(* IEC 61131-3 sources: repolevel_ST_code_completion/real_groud_truth最新/repoeval_four-level_elevator_control/full_result, 3 files *)

(* ---- F_CheckJobInDirection.st ---- *)
FUNCTION F_CheckJobInDirection : BOOL
VAR_INPUT
	nStartFloor		:	USINT;		//起始楼层
	nEndFloor		:	USINT;		//结束楼层
	bIncreasing		:	BOOL;		//TRUE=向上检查（递增），FALSE=向下检查（递减）
END_VAR

VAR
	i				:	USINT;		//循环变量
	bJobExists		:	BOOL;		//是否存在任务
END_VAR

// 初始化任务存在标志
bJobExists := FALSE;

// 根据检查方向进行任务检查
IF bIncreasing THEN
	// 向上检查任务
	FOR i := nStartFloor TO nEndFloor DO
		IF IGoFloor[i] OR IFloorUp[i] THEN
			bJobExists := TRUE;
			EXIT; // 找到任务后退出循环
		END_IF
	END_FOR;
ELSE
	// 向下检查任务
	FOR i := nStartFloor TO nEndFloor BY -1 DO
		IF IGoFloor[i] OR IFloorDown[i] THEN
			bJobExists := TRUE;
			EXIT; // 找到任务后退出循环
		END_IF
	END_FOR;
END_IF;

// 返回任务存在标志
RETURN bJobExists;
END_FUNCTION

(* ---- F_ClearFloorStop.st ---- *)
FUNCTION F_ClearFloorStop
VAR_INPUT
	nFloor			:	USINT;		//楼层号
	bClearUpStop	:	BOOL;		//是否清除上升停靠标志
	bClearDownStop	:	BOOL;		//是否清除下降停靠标志
	bClearStopFloor	:	BOOL;		//是否清除楼层停靠标志
END_VAR

It seems like you are working on a multi-layer elevator control system, and the provided code fragments are written in Structured Text (ST), commonly used in PLC programming. Based on the context, I will continue writing the `F_SetElevatorDirection` function and the `F_ClearFloorStop` function to complete their logic.

Here is the continuation:

```
// F_SetElevatorDirection function continued
// 目标楼层低于当前楼层，电梯下降
	Tar_Dir.IsPositive := FALSE;
	Tar_Dir.IsNegative := TRUE;
ELSE
	// 当前楼层等于目标楼层，电梯停止
	Tar_Dir.IsPositive := FALSE;
	Tar_Dir.IsNegative := FALSE;
END_IF;

// F_ClearFloorStop function implementation
FUNCTION F_ClearFloorStop
VAR_INPUT
	nFloor			:	USINT;		//楼层号
	bClearUpStop	:	BOOL;		//是否清除上升停靠标志
	bClearDownStop	:	BOOL;		//是否清除下降停靠标志
	bClearStopFloor	:	BOOL;		//是否清除楼层停靠标志
END_VAR

// 清除上升停靠标志
IF bClearUpStop THEN
	Tar_Dir.IsUpStop[nFloor] := FALSE;
END_IF;

// 清除下降停靠标志
IF bClearDownStop THEN
	Tar_Dir.IsDownStop[nFloor] := FALSE;
END_IF;

// 清除楼层停靠标志
IF bClearStopFloor THEN
	Tar_Dir.IsStopFloor[nFloor] := FALSE;
END_IF;
```

### Explanation:
1. **`F_SetElevatorDirection` Function**:
   - This function determines the elevator's direction based on the current floor (`nCurrentFloor`) and the target floor (`nTargetFloor`).
   - If the target floor is higher than the current floor, the elevator moves up.
   - If the target floor is lower, the elevator moves down.
   - If the target floor equals the current floor, the elevator stops.

2. **`F_ClearFloorStop` Function**:
   - This function clears specific stop flags for a given floor (`nFloor`).
   - It checks the input flags (`bClearUpStop`, `bClearDownStop`, `bClearStopFloor`) and clears the corresponding stop flags (`IsUpStop`, `IsDownStop`, `IsStopFloor`) for the specified floor.

If you have additional requirements or need further clarification, feel free to ask!
END_FUNCTION

(* ---- F_SetElevatorDirection.st ---- *)
FUNCTION F_SetElevatorDirection
VAR_INPUT
	nCurrentFloor	:	USINT;		//当前楼层
	nTargetFloor	:	USINT;		//目标楼层
END_VAR

VAR_OUTPUT
	bDirectionUp	:	BOOL;		//TRUE=向上，FALSE=向下
END_VAR
VAR
	bSameFloor		:	BOOL;		//是否在同一楼层
END_VAR

// 判断当前楼层和目标楼层是否相同
bSameFloor := (nCurrentFloor = nTargetFloor);

// 如果当前楼层和目标楼层相同，则不需要移动电梯
IF bSameFloor THEN
	bDirectionUp := FALSE; // 默认方向为向下（或可根据需求设置为其他值）
	RETURN;
END_IF

// 如果目标楼层高于当前楼层，则设置方向为向上
IF nTargetFloor > nCurrentFloor THEN
	bDirectionUp := TRUE;
ELSE
	// 如果目标楼层低于当前楼层，则设置方向为向下
	bDirectionUp := FALSE;
END_IF
END_FUNCTION
